(* PLC project Unnamed, Unknown Unnamed 1 *)
(* stored: creationDateTime 2026-03-18T20:32:34, modificationDateTime 2026-03-18T20:32:34 *)

PROGRAM main
  VAR
    Lid_at_place AT %IX100.0 : BOOL;  (* pokrywka przed zaciskiem *)
    Lid_clamped AT %IX100.1 : BOOL;
    Base_at_place AT %IX100.2 : BOOL;
    Base_clamped AT %IX100.3 : BOOL;
    Moving_X AT %IX100.4 : BOOL;
    Moving_Z AT %IX100.5 : BOOL;
    Item_detected AT %IX100.6 : BOOL;  (* Grabbed sucesfully *)
    Part_leaving AT %IX100.7 : BOOL;
    Lids_conveyor AT %QX100.0 : BOOL;
    Clamp_lid AT %QX100.1 : BOOL;  (* zacisnij *)
    Pos_raise_lid AT %QX100.2 : BOOL;
    Base_conveyor AT %QX100.3 : BOOL;
    Clamp_base AT %QX100.4 : BOOL;
    Move_X AT %QX100.5 : BOOL;
    Move_Z AT %QX100.6 : BOOL;
    Grab AT %QX100.7 : BOOL;
    Start AT %IX101.0 : BOOL;
  END_VAR
  VAR
    Delay : TIME := T#500ms;
    TON0 : TON;
    TOF0 : TOF;
    TOF1 : TOF;
    TON3 : TON;
    TOF2 : TON;
  END_VAR

(* LD diagram, written out as Structured Text *)
IF Start THEN Lids_conveyor := TRUE; END_IF;
IF Start THEN Clamp_lid := FALSE; END_IF;
TON3(IN := Lid_at_place OR Lid_clamped, PT := Delay);
IF TON3.Q THEN Lids_conveyor := FALSE; END_IF;
TOF2(IN := Lid_at_place, PT := Delay);
IF TOF2.Q THEN Clamp_lid := TRUE; END_IF;
END_PROGRAM

CONFIGURATION Config0
  RESOURCE Res0 ON PLC
    TASK task0(INTERVAL := T#20ms, PRIORITY := 1);
    PROGRAM instance0 WITH task0 : main;
  END_RESOURCE
END_CONFIGURATION
